Staubli VAL3: onF2Event.pgx

program onF2Event(bool& x_bSave[] (dimensions=1))
begin
  // look if the bButton is enable
  if bButton[1]
    //
    // CHANGE THE settings
    //
    setTextMode(1)
    call use:type(0,4,"F2 "+sMenu[1])
    setTextMode(0)
    call settings()
    use:bUseRefresh=true
    x_bSave=true
  endIf
end
